# EPICS substitutions: siteApps/EtherCat/m-epics-ecat2db/db/ecat2el1014.substitutions
file ecat2slave.template
{
	pattern {DEVICENAME}
		{EL1014}
}

file ecat2el10xxel11xxDI.template
{
	pattern {CH_ID, PDO_IDX}
		{$(MOD_ID)-DI1, 0}
		{$(MOD_ID)-DI2, 1}
		{$(MOD_ID)-DI3, 2}
		{$(MOD_ID)-DI4, 3}
}
